{attribute 'GeneratedUsingTerminal: BK1150-0000-0018'}
{attribute addProperty BoxType "BK1150-0000-0018"}
{attribute addProperty Id "Term_385_KL1002KL1002_BB38DA8F0"}
{attribute addProperty CRC "1764918420"}
{attribute addProperty Size "0"}
TYPE A_0012_BK1150_0000_0018_69328494 EXTENDS BK1150_A2FCADE7 :
STRUCT
	{attribute addProperty Name "Term_385_KL1002"}
	Term_385_KL1002 : KL1002_BB38DA8F;
END_STRUCT
END_TYPE

(* stored: Version 1.2.0.0, ProductVersion 3.1.4024.9
   DUT A_0012_BK1150_0000_0018_69328494: Id {bcad06b1-7b90-4c54-aad9-1dabe32e8632} *)
